{attribute 'GeneratedUsingTerminal: EL6695-0002-0001'}
{attribute addProperty BoxType "EL6695-0002-0001"}
{attribute addProperty Id "TxPDO_toggleAT %I*BOOL1TxPDO_stateAT %I*BOOL1External_device_not_connectedAT %I*BOOL1"}
{attribute addProperty CRC "501652368"}
{attribute addProperty Size "3"}
TYPE SYNC_Inputs_1DE69B90 :
STRUCT
	{attribute addProperty Name "TxPDO_toggle"}
	TxPDO_toggle AT %I* : BOOL;
	{attribute addProperty Name "TxPDO_state"}
	TxPDO_state AT %I* : BOOL;
	{attribute addProperty Name "External_device_not_connected"}
	External_device_not_connected AT %I* : BOOL;
END_STRUCT
END_TYPE

(* stored: Version 1.2.0.0, ProductVersion 3.1.4024.9
   DUT SYNC_Inputs_1DE69B90: Id {af7e1d57-0699-40f1-86ae-7025c257a4ad} *)
